{attribute 'linkalways'} 
{attribute 'no_explicit_call' := 'This FB is a CLASS and must be accessed using methods or properties'}
{attribute 'enable_dynamic_creation'}
FUNCTION_BLOCK Node_F_VN_MedianElementElementwise_TcVnVector4_UINT EXTENDS VisionNode
VAR
    ipContainer : _ITcVnContainer;
    aMedian : _TcVnVector4_UINT;
    hrPrev : _HRESULT(S_OK);
    hresult : _HRESULT(S_OK);
END_VAR

METHOD PUBLIC  Clone : I_Node
VAR
	pNode : POINTER TO Node_F_VN_MedianElementElementwise_TcVnVector4_UINT;
END_VAR
pNode := __NEW(Node_F_VN_MedianElementElementwise_TcVnVector4_UINT);
Clone := pNode^;
END_METHOD

METHOD FB_init : BOOL
VAR_INPUT
	bInitRetains : BOOL; // if TRUE, the retain variables are initialized (warm start / cold start)
	bInCopyCode : BOOL;  // if TRUE, the instance afterwards gets moved into the copy code (online change)
END_VAR
AddInput('ipContainer', ipContainer);
AddInput('aMedian', aMedian);
AddInput('hrPrev', hrPrev);
AddOutput('ipContainer', ipContainer);
AddOutput('hresult',hresult);
END_METHOD

METHOD PROTECTED OnExecute : HRESULT
hresult.Value := F_VN_MedianElementElementwise_TcVnVector4_UINT(
    ipContainer := ipContainer.Value,
    aMedian := aMedian.Value,
    hrPrev:= hrPrev.Value);
END_METHOD

METHOD PUBLIC PreExecutionCheck
VAR_INPUT
	Check : I_PreExecutionChecks;
END_VAR
Check.IsTrue(ipContainer.IsValid, 'ipContainer must be a valid container');
END_METHOD

END_FUNCTION_BLOCK

(* stored: Version 1.1.0.1, ProductVersion 3.1.4024.13
   POU Node_F_VN_MedianElementElementwise_TcVnVector4_UINT: Id {c6da301c-b21e-44dd-b086-8e114ba0a916}, SpecialFunc None
   Folder Constructor: Id {ec99388c-34ca-436a-85fe-dbef01bfde8b}
   Method Clone: Id {9b84f1b9-4fc6-4b5d-a44f-3d6898280b33}
   Method FB_init: Id {e49ff4db-d1e2-4f71-ab02-91cf19b11c77}
   Method OnExecute: Id {71979c5e-56be-49ef-9703-64107ac21c38}
   Method PreExecutionCheck: Id {76c9d5b9-995f-469c-8432-f61f6ec9ddc3} *)
